(* CODESYS project Untitled1.project

Project tree, tasks and I/O mapping:
  Device : CODESYS Control Win V3, 3S - Smart Software Solutions GmbH, order no. 305021, version 3.5.11.30
    application Application
      libraries: Standard, * (System)
      task MainTask (cyclic, interval t#20ms, priority 1) calls PLC_PRG
      program PLC_PRG [ST]
      function block FBMotor [ST]
*)

// Device/Application/PLC_PRG
PROGRAM PLC_PRG
VAR
	bt: BOOL ;
	aux: BOOL;
	vel: REAL := 1800;
	tensao: REAL := 220;
	deg: REAL := 22;
	
	btT: R_TRIG;
	q1T: R_TRIG;
	q2T: R_TRIG;
	
	out: REAL;
	
	T1: TP;
	TIME1: TIME;
	Q1: BOOL;
	
	T2: TOf;
	TIME2: TIME;
	Q2: BOOL;
	
	pass: REAL;
	
	
END_VAR

btT(clk:=bt);
q1T(clk:=NOT(q1));
q2T(clk:= NOT(q2));

pass := tensao/deg;

t1(in:= btT.Q OR q2t.q, pt:= T#1S, et=>time1, q=>q1);
t2(in:= q1T.Q, pt:= T#1S, et=>time1, q=>q2);

IF out < 220 THEN
	IF q1 THEN 
		aux:= TRUE;
	END_IF
	
	IF aux THEN 
		out := out + pass;
		aux:= FALSE;
	END_IF
	
	IF q2 THEN 
		q1 := FALSE;
	END_IF
END_IF

END_PROGRAM

// Device/Application/FBMotor
FUNCTION_BLOCK FBMotor
VAR_INPUT
	R1: R_TRIG;
	tensao: REAL;
	vel: REAL;
	deg: INT;
	bt1: BOOL;
END_VAR
VAR_OUTPUT
	out: REAL;
END_VAR
VAR
	cont: INT;
	t1: TOF;
	AUX: BOOL;
	time1: TIME;
	q1: BOOL;
	ifcont: INT;
	divten: REAL;
	divvel: REAL;
	value: REAL:= 0.0;
	Q: BOOL;
END_VAR

divten:= tensao/deg;
divvel:= vel/deg;

IF bt1 THEN
	AUX:=TRUE;
END_IF

IF aux THEN
	t1(in:=,pt:=T#1S,et=>time1,q =>q1);
	out := value + divten;
	cont := cont +1;
END_IF


R1(CLK:=NOT(AUX));

END_FUNCTION_BLOCK
